FUNCTION F_DegPerMinToDegPerSec : LREAL
VAR_INPUT
	fValue : LREAL; // °/min value
END_VAR
VAR
END_VAR

 F_DegPerMinToDegPerSec := fValue/60; // °/min -> °/s

END_FUNCTION

(* stored: Version 1.1.0.1, ProductVersion 3.1.4024.12
   POU F_DegPerMinToDegPerSec: Id {99ac8d63-0783-4291-a09e-5eb3394a3ceb}, SpecialFunc None *)
